// TIA Portal project "Project2" (V16)

(* hardware
DEVICE "S7-1200 station_1"  S7-1200 Station
   slot 0: "Rack_0"  S7-1200 Rack  Rack  V1.0
   slot 1: "1214C"  CPU 1214C AC/DC/Rly  6ES7 214-1BG31-0XB0  V3.0
   slot 2: "AI 4x13BIT_1"  SM 1231 AI4  6ES7 231-4HD30-0XB0  V1.0
   slot 3: "DI 16x24VDC_1"  SM 1221 DI16 x 24VDC  6ES7 221-1BH30-0XB0  V1.0
   slot 4: "AQ 4x14BIT_1"  SM 1232 AQ4  6ES7 232-4HD30-0XB0  V1.0
*)

// ===== PLC "1214C"  CPU 1214C AC/DC/Rly =====

VAR_GLOBAL   // PLC tag table "Default tag table"
   "Level Switch in Water Tank" AT %I0.0 : Bool;
   "Auto Selection" AT %I0.2 : Bool;
   "Manual Selection" AT %I0.3 : Bool;
   "Auto Start Push Button" AT %I0.4 : Bool;
   "Auto Stop Push Button" AT %I0.5 : Bool;
   "Conveyor Start in Manual Mode" AT %I0.6 : Bool;
   "Conveyor Stop in Manual Mode" AT %I0.7 : Bool;
   "Proximity Sensor for Bottle Filling" AT %I0.1 : Bool;
   "SV Stop in Manual Mode" AT %I1.1 : Bool;
   "Emergency Switch" AT %I1.2 : Bool;
   "SV Open CMD" AT %Q0.1 : Bool;
   "Conveyor Start Indication" AT %Q0.2 : Bool;
   "Conveyor Start CMD" AT %Q0.0 : Bool;
   "SV Open Indication" AT %Q0.3 : Bool;
   "Water Pump" AT %Q0.4 : Bool;
   "Tag_1" AT %M0.0 : Bool;
   "Tag_2" AT %M0.1 : Bool;
   "Tag_3" AT %M0.3 : Bool;
   "Tag_4" AT %M0.2 : Bool;
   "SV START IN MANUAL MODE" AT %I1.0 : Bool;
END_VAR

DATA_BLOCK "Data_block_1"   // DB2
{ S7_Optimized_Access := 'TRUE' }
VERSION : 0.1
// stored: InstanceOfName Block_1
"Block_1"
BEGIN
END_DATA_BLOCK

DATA_BLOCK "Block_1_DB"   // DB3
{ S7_Optimized_Access := 'TRUE' }
VERSION : 0.1
// stored: InstanceOfName Block_1
"Block_1"
BEGIN
END_DATA_BLOCK

// folder: System blocks/Program resources

DATA_BLOCK "IEC_Timer_0_DB"   // DB1
{ S7_Optimized_Access := 'TRUE' }
AUTHOR : Simatic
FAMILY : IEC
NAME : IEC_TMR
VERSION : 1.0
// stored: InstanceOfName IEC_TIMER
"IEC_TIMER"
BEGIN
END_DATA_BLOCK

// folder: (top level)

FUNCTION_BLOCK "Block_1"   // FB1, LAD
{ S7_Optimized_Access := 'TRUE' }
VERSION : 0.1
   VAR_TEMP   // added for the SCL form of the ladder/FBD networks
      _w1 : Bool;
      _w2 : Bool;
   END_VAR
BEGIN

REGION Network 1
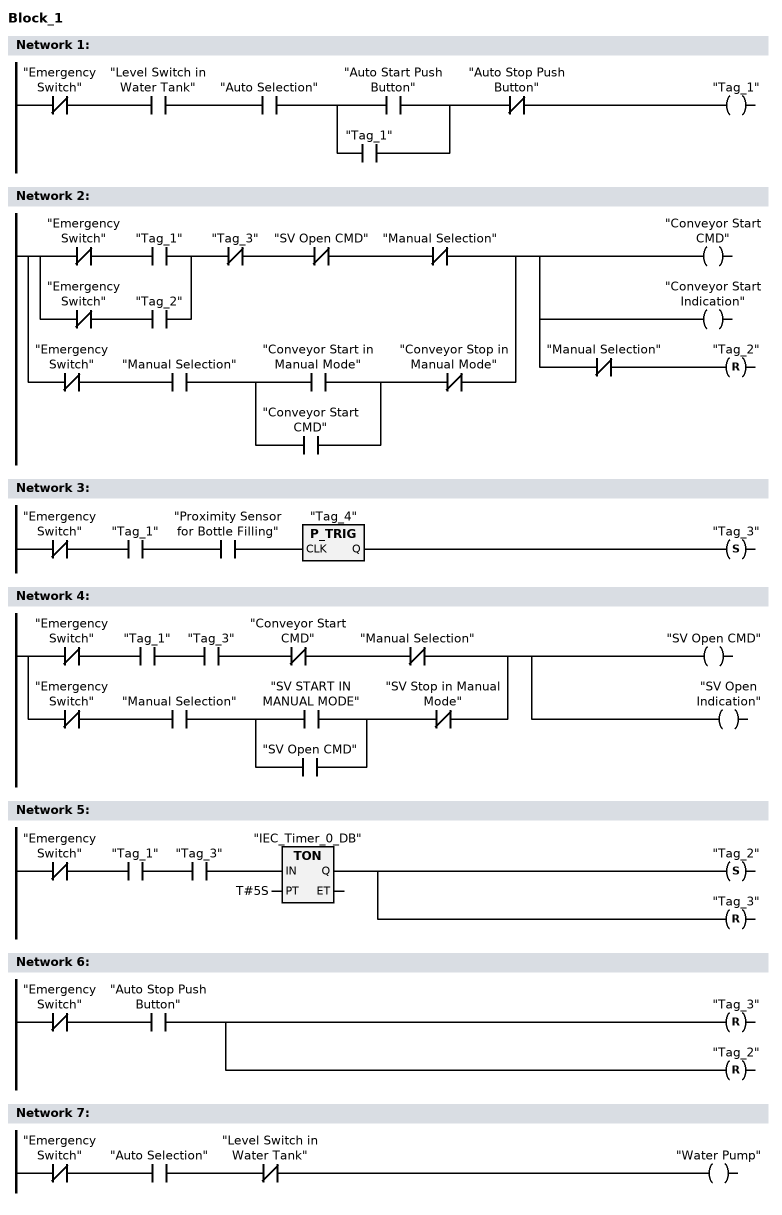
   RUNG wire#powerrail
      I_Contact( "Emergency Switch" )
      Contact( "Level Switch in Water Tank" )
      Contact( "Auto Selection" )
      wire#w1
      Contact( "Auto Start Push Button" )
      wire#w2
      I_Contact( "Auto Stop Push Button" )
      Coil( "Tag_1" )
   END_RUNG
   RUNG wire#w1
      Contact( "Tag_1" )
   END_RUNG wire#w2
   // the same network as SCL:
   "Tag_1" := NOT "Emergency Switch" AND "Level Switch in Water Tank" AND "Auto Selection" AND ("Auto Start Push Button" OR "Tag_1") AND NOT "Auto Stop Push Button";
END_REGION

REGION Network 2
   RUNG wire#powerrail
      I_Contact( "Emergency Switch" )
      Contact( "Tag_1" )
      wire#w1
      I_Contact( "Tag_3" )
      I_Contact( "SV Open CMD" )
      I_Contact( "Manual Selection" )
      wire#w2
      Coil( "Conveyor Start CMD" )
   END_RUNG
   RUNG wire#powerrail
      I_Contact( "Emergency Switch" )
      Contact( "Tag_2" )
   END_RUNG wire#w1
   RUNG wire#powerrail
      I_Contact( "Emergency Switch" )
      Contact( "Manual Selection" )
      wire#w3
      Contact( "Conveyor Start in Manual Mode" )
      wire#w4
      I_Contact( "Conveyor Stop in Manual Mode" )
   END_RUNG wire#w2
   RUNG wire#w3
      Contact( "Conveyor Start CMD" )
   END_RUNG wire#w4
   RUNG wire#w2
      Coil( "Conveyor Start Indication" )
   END_RUNG
   RUNG wire#w2
      I_Contact( "Manual Selection" )
      R_Coil( "Tag_2" )
   END_RUNG
   // the same network as SCL:
   "Conveyor Start CMD" := (((NOT "Emergency Switch" AND "Tag_1") OR (NOT "Emergency Switch" AND "Tag_2")) AND NOT "Tag_3" AND NOT "SV Open CMD" AND NOT "Manual Selection") OR (NOT "Emergency Switch" AND "Manual Selection" AND ("Conveyor Start in Manual Mode" OR "Conveyor Start CMD") AND NOT "Conveyor Stop in Manual Mode");
   "Conveyor Start Indication" := "Conveyor Start CMD";
   IF "Conveyor Start CMD" AND NOT "Manual Selection" THEN "Tag_2" := FALSE; END_IF;
END_REGION

REGION Network 3
   RUNG wire#powerrail
      I_Contact( "Emergency Switch" )
      Contact( "Tag_1" )
      Contact( "Proximity Sensor for Bottle Filling" )
      P_Trig( "Tag_4" )
      S_Coil( "Tag_3" )
   END_RUNG
   // the same network as SCL:
   #_w1 := NOT "Emergency Switch" AND "Tag_1" AND "Proximity Sensor for Bottle Filling";
   #_w2 := #_w1 AND NOT "Tag_4";   // rising edge
   "Tag_4" := #_w1;
   IF #_w2 THEN "Tag_3" := TRUE; END_IF;
END_REGION

REGION Network 4
   RUNG wire#powerrail
      I_Contact( "Emergency Switch" )
      Contact( "Tag_1" )
      Contact( "Tag_3" )
      I_Contact( "Conveyor Start CMD" )
      I_Contact( "Manual Selection" )
      wire#w1
      Coil( "SV Open CMD" )
   END_RUNG
   RUNG wire#powerrail
      I_Contact( "Emergency Switch" )
      Contact( "Manual Selection" )
      wire#w2
      Contact( "SV START IN MANUAL MODE" )
      wire#w3
      I_Contact( "SV Stop in Manual Mode" )
   END_RUNG wire#w1
   RUNG wire#w2
      Contact( "SV Open CMD" )
   END_RUNG wire#w3
   RUNG wire#w1
      Coil( "SV Open Indication" )
   END_RUNG
   // the same network as SCL:
   "SV Open CMD" := (NOT "Emergency Switch" AND "Tag_1" AND "Tag_3" AND NOT "Conveyor Start CMD" AND NOT "Manual Selection") OR (NOT "Emergency Switch" AND "Manual Selection" AND ("SV START IN MANUAL MODE" OR "SV Open CMD") AND NOT "SV Stop in Manual Mode");
   "SV Open Indication" := "SV Open CMD";
END_REGION

REGION Network 5
   "IEC_Timer_0_DB".TON(IN := NOT "Emergency Switch" AND "Tag_1" AND "Tag_3", PT := T#5S);
   IF "IEC_Timer_0_DB".Q THEN
       "Tag_2" := TRUE;
       "Tag_3" := FALSE;
   END_IF;
END_REGION

REGION Network 6
   RUNG wire#powerrail
      I_Contact( "Emergency Switch" )
      Contact( "Auto Stop Push Button" )
      wire#w1
      R_Coil( "Tag_3" )
   END_RUNG
   RUNG wire#w1
      R_Coil( "Tag_2" )
   END_RUNG
   // the same network as SCL:
   IF NOT "Emergency Switch" AND "Auto Stop Push Button" THEN
       "Tag_3" := FALSE;
       "Tag_2" := FALSE;
   END_IF;
END_REGION

REGION Network 7
   RUNG wire#powerrail
      I_Contact( "Emergency Switch" )
      Contact( "Auto Selection" )
      I_Contact( "Level Switch in Water Tank" )
      Coil( "Water Pump" )
   END_RUNG
   // the same network as SCL:
   "Water Pump" := NOT "Emergency Switch" AND "Auto Selection" AND NOT "Level Switch in Water Tank";
END_REGION
END_FUNCTION_BLOCK

ORGANIZATION_BLOCK "Main"   // OB1, LAD, ProgramCycle
TITLE = "Main Program Sweep (Cycle)"
{ S7_Optimized_Access := 'TRUE' }
VERSION : 0.1
BEGIN

REGION Network 1
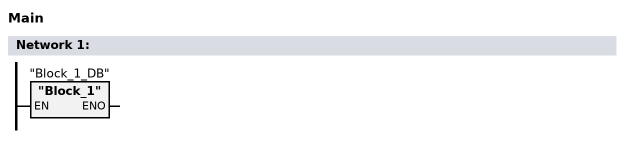
   RUNG wire#powerrail
      "Block_1_DB"()
   END_RUNG
   // the same network as SCL:
   "Block_1_DB"();   // "Block_1"
END_REGION
END_ORGANIZATION_BLOCK